KUKA KRL program: search.src, search.dat

--- search.src ---
&ACCESS RVP
&REL 7
&PARAM DISKPATH = KRC:\R1\Program
DEF  search ( )
   ;FOLD INI;%{PE}
      ;FOLD BASISTECH INI
         GLOBAL INTERRUPT DECL 3 WHEN $STOPMESS==TRUE DO IR_STOPM ( )
         INTERRUPT ON 3
         BAS (#INITMOV,0 )
      ;ENDFOLD (BASISTECH INI)
      ;FOLD USER INI
         ;Make your modifications here

      ;ENDFOLD (USER INI)
   ;ENDFOLD (INI)

;reset counter for program reset
ccount = 0

;define interrupt
   interrupt decl 99 when $in[27]==true do foundcube()

   ;FOLD PTP HOME  Vel= 100 % DEFAULT;%{PE}%MKUKATPBASIS,%CMOVE,%VPTP,%P 1:PTP, 2:HOME, 3:, 5:100, 7:DEFAULT
      $BWDSTART = FALSE
      PDAT_ACT=PDEFAULT
      FDAT_ACT=FHOME
      BAS (#PTP_PARAMS,100 )
      $H_POS=XHOME
      PTP  XHOME
   ;ENDFOLD
 interrupt on 99
   wait sec 0
   eyeson()

;FOLD PTP startscan Vel=100 % PDAT1 Tool[15]:DEMO_GRIPPER Base[1]:bluetable;%{PE}%R 8.3.34,%MKUKATPBASIS,%CMOVE,%VPTP,%P 1:PTP, 2:startscan, 3:, 5:100, 7:PDAT1
$BWDSTART=FALSE
PDAT_ACT=PPDAT1
FDAT_ACT=Fstartscan
BAS(#PTP_PARAMS,100)
PTP Xstartscan
;ENDFOLD


;FOLD LIN endscan CONT Vel=1 m/s CPDAT1 Tool[15]:DEMO_GRIPPER Base[1]:bluetable;%{PE}%R 8.3.34,%MKUKATPBASIS,%CMOVE,%VLIN,%P 1:LIN, 2:endscan, 3:C_DIS C_DIS, 5:1, 7:CPDAT1
$BWDSTART=FALSE
LDAT_ACT=LCPDAT1
FDAT_ACT=Fendscan
BAS(#CP_PARAMS,1)
LIN Xendscan C_DIS C_DIS
;ENDFOLD
   wait sec 0
   eyesoff()
   interrupt off 99

   ;move back to scan position
   $APO.cdis = 300
   ptp xstartscan c_dis

   ;move to scanned positions
   for ccount = 1 to 3
      ptp cubepos[1,ccount]
      wait sec 0.2
   endfor

   ;FOLD PTP HOME  Vel= 100 % DEFAULT;%{PE}%MKUKATPBASIS,%CMOVE,%VPTP,%P 1:PTP, 2:HOME, 3:, 5:100, 7:DEFAULT
      $BWDSTART = FALSE
      PDAT_ACT=PDEFAULT
      FDAT_ACT=FHOME
      BAS (#PTP_PARAMS,100 )
      $H_POS=XHOME
      PTP  XHOME
   ;ENDFOLD
END

def eyeson()
   $out[27] = true
end

def eyesoff()
   $out[27] = false
end

def foundcube()
decl KRLMSG_T mymessage
decl KRLMSGPAR_T params[3]
decl KRLMSGOPT_T opts
decl int hh
decl EKRLMSGTYPE headsup

   interrupt off

;iterate counter
ccount = ccount + 1

;display current pos x,y,z

;fold Message: Cube detected at position X,Y,Z
   headsup = #notify
   mymessage={modul[] "College", Nr 1999, msg_txt[] "Cube detected! X: %1 Y: %2 Z: %3"}
   opts = {VL_STOP true, CLEAR_P_RESET true, clear_p_saw false, log_to_db true}
   ;params / placeholder
   params[1] = {par_type #value}
   params[1].par_int = $POS_INT.x
   params[2] = {par_type #value}
   params[2].par_int = $POS_INT.y
   params[3] = {par_type #value}
   params[3].par_int = $POS_INT.z

   cubepos[1,ccount] = $pos_int
   ;generate message
   hh = set_krlmsg(headsup, mymessage, params[], opts)
;endfold

   interrupt on 99

end

--- search.dat ---
&ACCESS RVP
&REL 7
&PARAM DISKPATH = KRC:\R1\Program
DEFDAT  search
;FOLD EXTERNAL DECLARATIONS;%{PE}%MKUKATPBASIS,%CEXT,%VCOMMON,%P
;FOLD BASISTECH EXT;%{PE}%MKUKATPBASIS,%CEXT,%VEXT,%P
EXT  BAS (BAS_COMMAND  :IN,REAL  :IN )
;ENDFOLD (BASISTECH EXT)
;FOLD USER EXT;%{E}%MKUKATPUSER,%CEXT,%VEXT,%P
;Make your modifications here

;ENDFOLD (USER EXT)
;ENDFOLD (EXTERNAL DECLARATIONS)
DECL E6POS cubepos[1,3]
DECL INT ccount=1

DECL BASIS_SUGG_T LAST_BASIS={POINT1[] "endscan                 ",POINT2[] "endscan                 ",CP_PARAMS[] "CPDAT1                  ",PTP_PARAMS[] "PDAT1                   ",CONT[] "C_DIS C_DIS             ",CP_VEL[] "1                       ",PTP_VEL[] "100                     ",SYNC_PARAMS[] "SYNCDAT                 ",SPL_NAME[] "S0                      ",A_PARAMS[] "ADAT0                   "}
DECL E6POS XSTARTSCAN={X 329.084869,Y 34.0443687,Z 147.065567,A -115.348572,B 89.8659058,C -115.369781,S 6,T 58,E1 0.0,E2 0.0,E3 0.0,E4 0.0,E5 0.0,E6 0.0}
DECL FDAT Fstartscan={TOOL_NO 15,BASE_NO 1,IPO_FRAME #BASE,POINT2[] " ",TQ_STATE FALSE}
DECL PDAT PPDAT1={VEL 100.000,ACC 100.000,APO_DIST 100.000,GEAR_JERK 50.0000,EXAX_IGN 0}
DECL E6POS XENDSCAN={X -35.5893059,Y 33.9097595,Z 147.431320,A -115.348587,B 89.8659058,C -115.369797,S 6,T 58,E1 0.0,E2 0.0,E3 0.0,E4 0.0,E5 0.0,E6 0.0}
DECL FDAT Fendscan={TOOL_NO 15,BASE_NO 1,IPO_FRAME #BASE,POINT2[] " ",TQ_STATE FALSE}
DECL LDAT LCPDAT1={VEL 2.00000,ACC 100.000,APO_DIST 100.000,APO_FAC 50.0000,AXIS_VEL 100.000,AXIS_ACC 100.000,ORI_TYP #VAR,CIRC_TYP #BASE,JERK_FAC 50.0000,GEAR_JERK 50.0000,EXAX_IGN 0}
ENDDAT
